(* Logix 5000 project; controller CarbonScout_MK6 vendor 1 type 14 code 154 rev 32.11; software revision 32.00; part 10 of 17 *)
(* tags used below, declared in another part *)
   Delay : TIMER;
   ExtraValveCNTReached : BOOL;
   i : DINT;
   LIT_Prev : REAL;
   LocalSampleTank : DINT;
   ONS : BOOL[32];
   TankDiagnosticCheck : BOOL;
   TimeCompare : TimerCompare;
   XRF_DirtyWinCounter : COUNTER;
   AI_FIT_01 : P_AIn;   // Purge water flow
   AI_LIT_01 : P_AIn;   // Carbon Scout Laser Level Transmitter
   AI_LIT_02 : P_AIn;   // Carbon Scout Cone Level Transmitter
   AI_PIT_01 : P_AIn;   // Water supply pressure
   CS_Alarms : P_Alarm[80];
   CS_DINTParams : DINT[100];
   CS_REALParams : REAL[80];   // CS REAL Parameters
   CS_Seq : GEK_Sequence;
   CS_Tank : CS_TankParams[20];
   CS_Timer : TIMER[80];
   CS_XRF : XRF;
   NetworkHealthy : DINT;
   Oneshot : DINT;
   Oneshot3 : DINT;
   TimeAndDate : DINT[7];
   Valve_SPR_01_Stats : GekkoValveStat;
   Valve_XV_01_Stats : GekkoValveStat;
   Valve_XV_02_Stats : GekkoValveStat;
   Valve_XV_03_Stats : GekkoValveStat;
   Valve_XV_04_Stats : GekkoValveStat;
   Valve_XV_05_Stats : GekkoValveStat;
   Valve_XV_06_Stats : GekkoValveStat;
   Valve_XV_07_Stats : GekkoValveStat;
   Valve_XV_08_Stats : GekkoValveStat;
   Valve_XV_09_Stats : GekkoValveStat;
   Valve_XV_10_Stats : GekkoValveStat;
   Valve_XV_11 : P_ValveSO;   // Purge Valve
   Valve_XV_11_Stats : GekkoValveStat;
   Valve_XV_12 : P_ValveSO;   // Slurry inlet vavle
   Valve_XV_12_Stats : GekkoValveStat;
   Valve_XV_13_Stats : GekkoValveStat;
   Valve_XV_14 : P_ValveSO;   // Top wash vavle
   Valve_XV_14_Stats : GekkoValveStat;
   Valve_XV_15_Stats : GekkoValveStat;
   Valve_XV_16_Stats : GekkoValveStat;
   Valve_XV_17 : P_ValveSO;   // Sample cone outlet vavle
   Valve_XV_17_Stats : GekkoValveStat;
   Valve_XV_18_Stats : GekkoValveStat;
   Valve_XV_19 : P_ValveSO;   // Laser window
   Valve_XV_19_Stats : GekkoValveStat;
   Valve_XV_21_30_Stats : GekkoValveStat;
   Valve_XV_30_Stats : GekkoValveStat;
   XRF_RAWDINT : DINT[100];
(* SeqProgram, continued *)

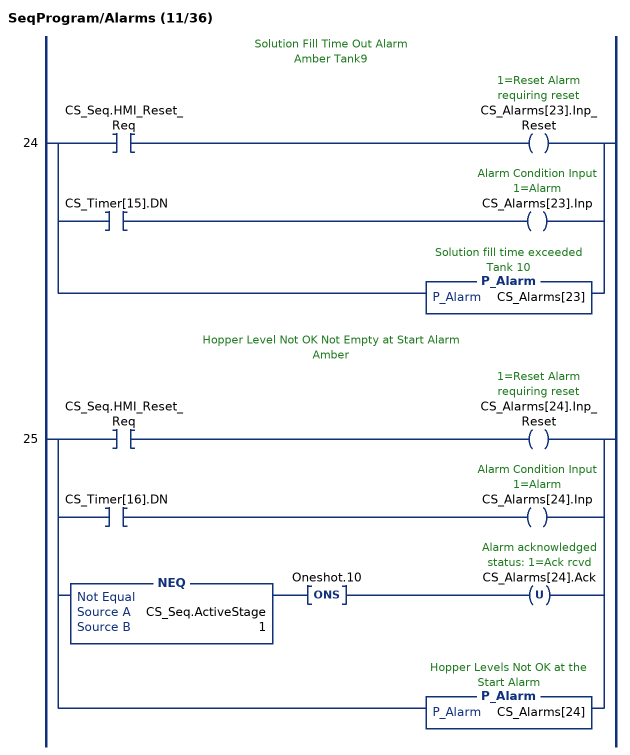
   // Solution Fill Time Out Alarm
   // Amber Tank9
   24: [XIC(CS_Seq.HMI_Reset_Req) OTE(CS_Alarms[23].Inp_Reset) ,XIC(CS_Timer[15].DN) OTE(CS_Alarms[23].Inp) ,P_Alarm(CS_Alarms[23]) ];
   // Hopper Level Not OK Not Empty at Start Alarm
   // Amber
   25: [XIC(CS_Seq.HMI_Reset_Req) OTE(CS_Alarms[24].Inp_Reset) ,XIC(CS_Timer[16].DN) OTE(CS_Alarms[24].Inp) ,NEQ(CS_Seq.ActiveStage,1) ONS(Oneshot.10) OTU(CS_Alarms[24].Ack) ,P_Alarm(CS_Alarms[24]) ];
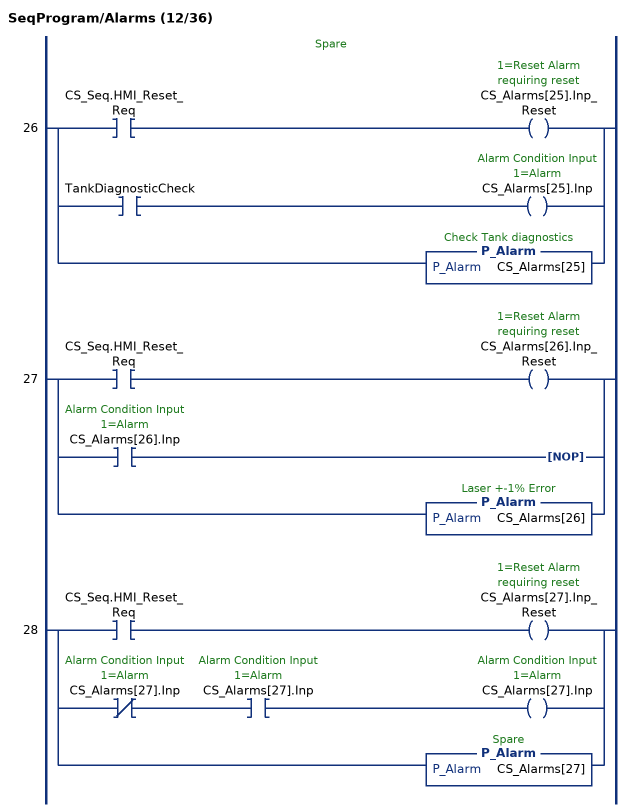
   // Spare
   26: [XIC(CS_Seq.HMI_Reset_Req) OTE(CS_Alarms[25].Inp_Reset) ,XIC(TankDiagnosticCheck) OTE(CS_Alarms[25].Inp) ,P_Alarm(CS_Alarms[25]) ];
   27: [XIC(CS_Seq.HMI_Reset_Req) OTE(CS_Alarms[26].Inp_Reset) ,XIC(CS_Alarms[26].Inp) NOP() ,P_Alarm(CS_Alarms[26]) ];
   28: [XIC(CS_Seq.HMI_Reset_Req) OTE(CS_Alarms[27].Inp_Reset) ,XIO(CS_Alarms[27].Inp) XIC(CS_Alarms[27].Inp) OTE(CS_Alarms[27].Inp) ,P_Alarm(CS_Alarms[27]) ];
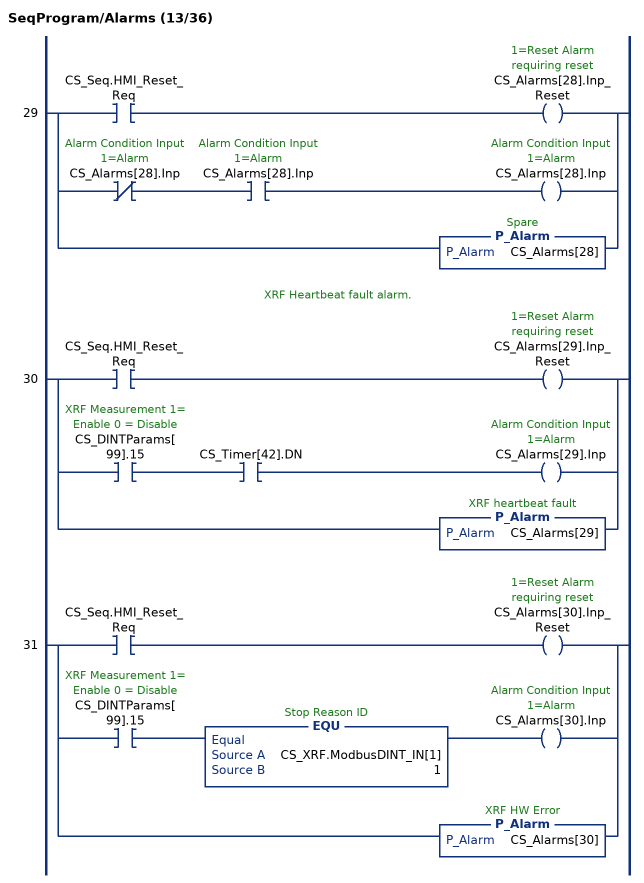
   29: [XIC(CS_Seq.HMI_Reset_Req) OTE(CS_Alarms[28].Inp_Reset) ,XIO(CS_Alarms[28].Inp) XIC(CS_Alarms[28].Inp) OTE(CS_Alarms[28].Inp) ,P_Alarm(CS_Alarms[28]) ];
   // XRF Heartbeat fault alarm.
   30: [XIC(CS_Seq.HMI_Reset_Req) OTE(CS_Alarms[29].Inp_Reset) ,XIC(CS_DINTParams[99].15) XIC(CS_Timer[42].DN) OTE(CS_Alarms[29].Inp) ,P_Alarm(CS_Alarms[29]) ];
   31: [XIC(CS_Seq.HMI_Reset_Req) OTE(CS_Alarms[30].Inp_Reset) ,XIC(CS_DINTParams[99].15) EQU(CS_XRF.ModbusDINT_IN[1],1) OTE(CS_Alarms[30].Inp) ,P_Alarm(CS_Alarms[30]) ];
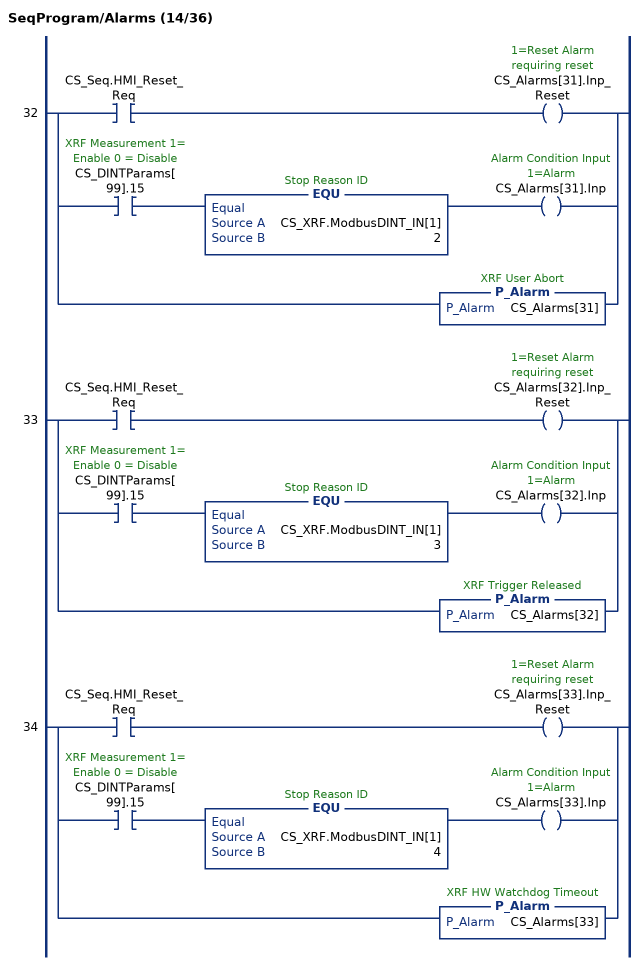
   32: [XIC(CS_Seq.HMI_Reset_Req) OTE(CS_Alarms[31].Inp_Reset) ,XIC(CS_DINTParams[99].15) EQU(CS_XRF.ModbusDINT_IN[1],2) OTE(CS_Alarms[31].Inp) ,P_Alarm(CS_Alarms[31]) ];
   33: [XIC(CS_Seq.HMI_Reset_Req) OTE(CS_Alarms[32].Inp_Reset) ,XIC(CS_DINTParams[99].15) EQU(CS_XRF.ModbusDINT_IN[1],3) OTE(CS_Alarms[32].Inp) ,P_Alarm(CS_Alarms[32]) ];
   34: [XIC(CS_Seq.HMI_Reset_Req) OTE(CS_Alarms[33].Inp_Reset) ,XIC(CS_DINTParams[99].15) EQU(CS_XRF.ModbusDINT_IN[1],4) OTE(CS_Alarms[33].Inp) ,P_Alarm(CS_Alarms[33]) ];
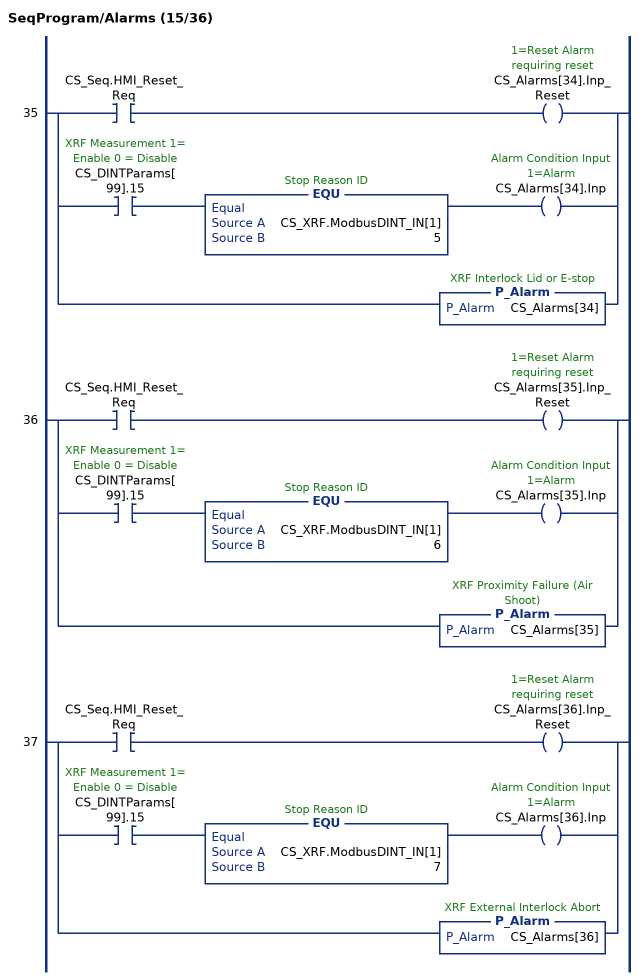
   35: [XIC(CS_Seq.HMI_Reset_Req) OTE(CS_Alarms[34].Inp_Reset) ,XIC(CS_DINTParams[99].15) EQU(CS_XRF.ModbusDINT_IN[1],5) OTE(CS_Alarms[34].Inp) ,P_Alarm(CS_Alarms[34]) ];
   36: [XIC(CS_Seq.HMI_Reset_Req) OTE(CS_Alarms[35].Inp_Reset) ,XIC(CS_DINTParams[99].15) EQU(CS_XRF.ModbusDINT_IN[1],6) OTE(CS_Alarms[35].Inp) ,P_Alarm(CS_Alarms[35]) ];
   37: [XIC(CS_Seq.HMI_Reset_Req) OTE(CS_Alarms[36].Inp_Reset) ,XIC(CS_DINTParams[99].15) EQU(CS_XRF.ModbusDINT_IN[1],7) OTE(CS_Alarms[36].Inp) ,P_Alarm(CS_Alarms[36]) ];
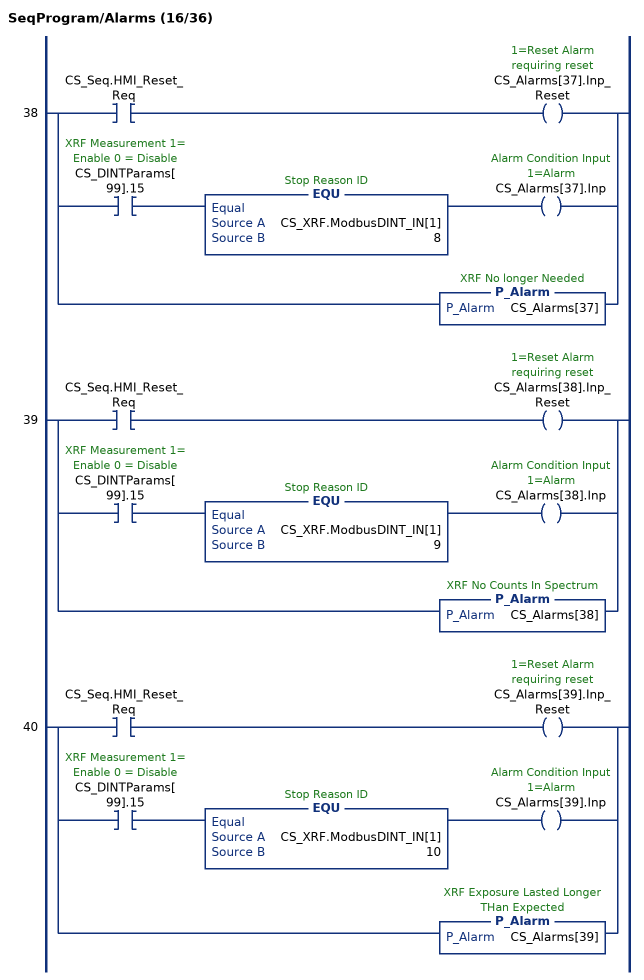
   38: [XIC(CS_Seq.HMI_Reset_Req) OTE(CS_Alarms[37].Inp_Reset) ,XIC(CS_DINTParams[99].15) EQU(CS_XRF.ModbusDINT_IN[1],8) OTE(CS_Alarms[37].Inp) ,P_Alarm(CS_Alarms[37]) ];
   39: [XIC(CS_Seq.HMI_Reset_Req) OTE(CS_Alarms[38].Inp_Reset) ,XIC(CS_DINTParams[99].15) EQU(CS_XRF.ModbusDINT_IN[1],9) OTE(CS_Alarms[38].Inp) ,P_Alarm(CS_Alarms[38]) ];
   40: [XIC(CS_Seq.HMI_Reset_Req) OTE(CS_Alarms[39].Inp_Reset) ,XIC(CS_DINTParams[99].15) EQU(CS_XRF.ModbusDINT_IN[1],10) OTE(CS_Alarms[39].Inp) ,P_Alarm(CS_Alarms[39]) ];
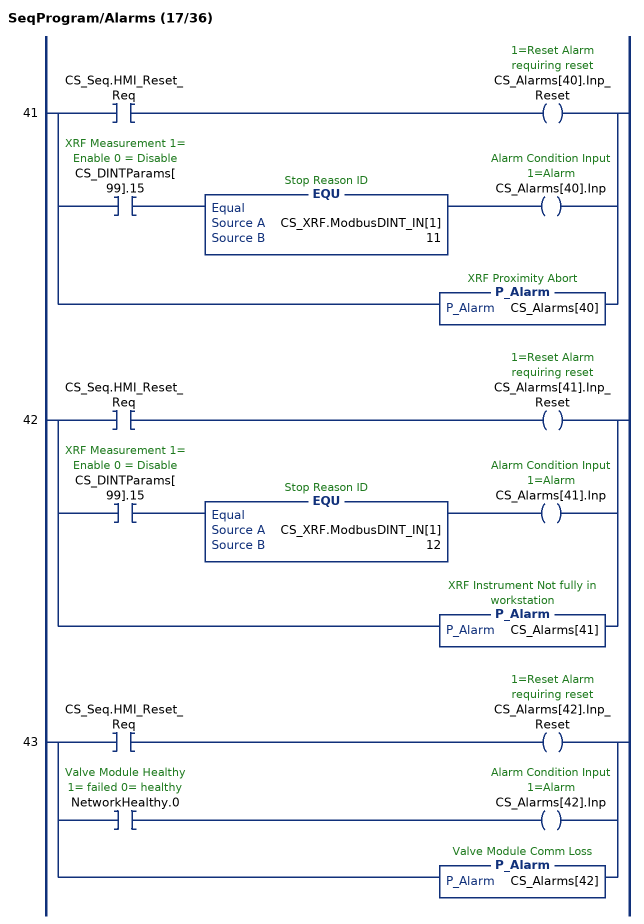
   41: [XIC(CS_Seq.HMI_Reset_Req) OTE(CS_Alarms[40].Inp_Reset) ,XIC(CS_DINTParams[99].15) EQU(CS_XRF.ModbusDINT_IN[1],11) OTE(CS_Alarms[40].Inp) ,P_Alarm(CS_Alarms[40]) ];
   42: [XIC(CS_Seq.HMI_Reset_Req) OTE(CS_Alarms[41].Inp_Reset) ,XIC(CS_DINTParams[99].15) EQU(CS_XRF.ModbusDINT_IN[1],12) OTE(CS_Alarms[41].Inp) ,P_Alarm(CS_Alarms[41]) ];
   43: [XIC(CS_Seq.HMI_Reset_Req) OTE(CS_Alarms[42].Inp_Reset) ,XIC(NetworkHealthy.0) OTE(CS_Alarms[42].Inp) ,P_Alarm(CS_Alarms[42]) ];
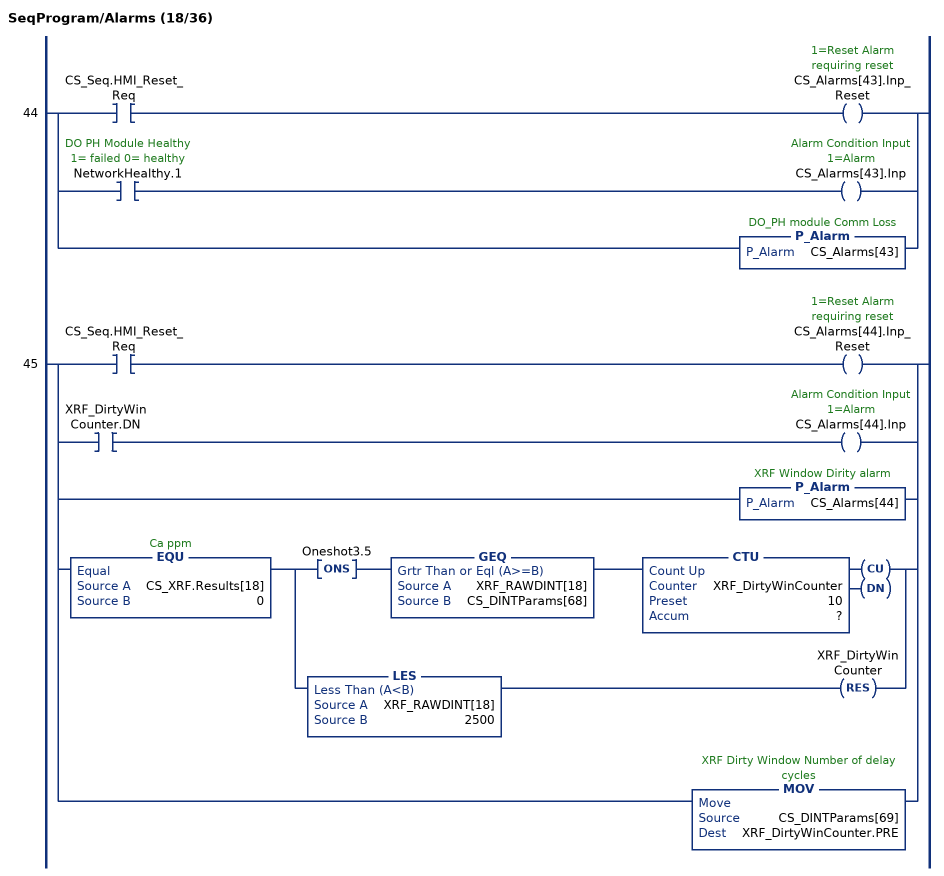
   44: [XIC(CS_Seq.HMI_Reset_Req) OTE(CS_Alarms[43].Inp_Reset) ,XIC(NetworkHealthy.1) OTE(CS_Alarms[43].Inp) ,P_Alarm(CS_Alarms[43]) ];
   45: [XIC(CS_Seq.HMI_Reset_Req) OTE(CS_Alarms[44].Inp_Reset) ,XIC(XRF_DirtyWinCounter.DN) OTE(CS_Alarms[44].Inp) ,P_Alarm(CS_Alarms[44]) ,EQU(CS_XRF.Results[18],0) [ONS(Oneshot3.5) GEQ(XRF_RAWDINT[18],CS_DINTParams[68]) CTU(XRF_DirtyWinCounter,?,?) ,LES(XRF_RAWDINT[18],2500) RES(XRF_DirtyWinCounter) ] ,MOV(CS_DINTParams[69],XRF_DirtyWinCounter.PRE) ];
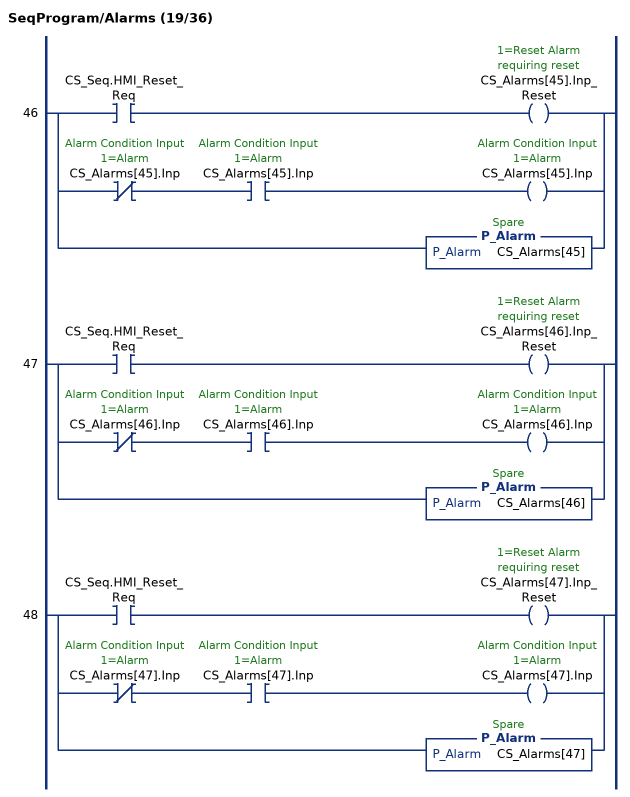
   46: [XIC(CS_Seq.HMI_Reset_Req) OTE(CS_Alarms[45].Inp_Reset) ,XIO(CS_Alarms[45].Inp) XIC(CS_Alarms[45].Inp) OTE(CS_Alarms[45].Inp) ,P_Alarm(CS_Alarms[45]) ];
   47: [XIC(CS_Seq.HMI_Reset_Req) OTE(CS_Alarms[46].Inp_Reset) ,XIO(CS_Alarms[46].Inp) XIC(CS_Alarms[46].Inp) OTE(CS_Alarms[46].Inp) ,P_Alarm(CS_Alarms[46]) ];
   48: [XIC(CS_Seq.HMI_Reset_Req) OTE(CS_Alarms[47].Inp_Reset) ,XIO(CS_Alarms[47].Inp) XIC(CS_Alarms[47].Inp) OTE(CS_Alarms[47].Inp) ,P_Alarm(CS_Alarms[47]) ];
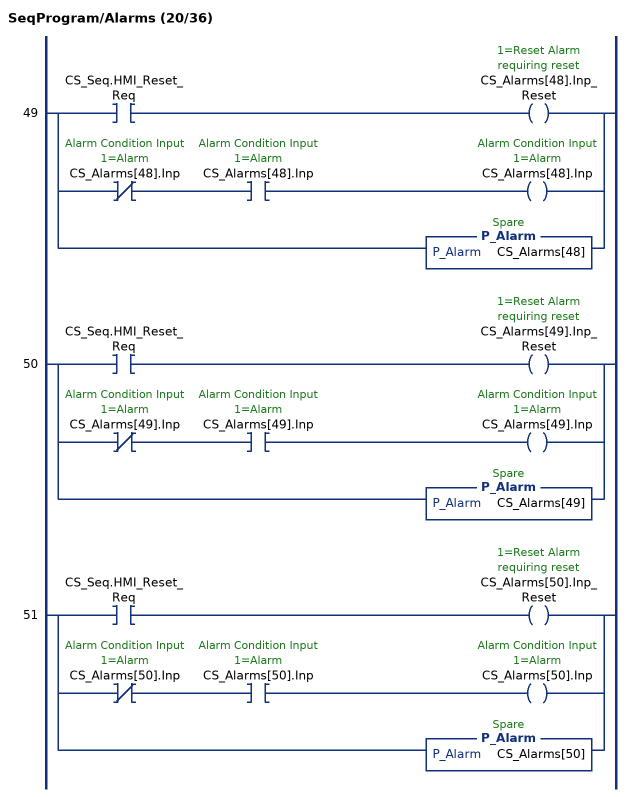
   49: [XIC(CS_Seq.HMI_Reset_Req) OTE(CS_Alarms[48].Inp_Reset) ,XIO(CS_Alarms[48].Inp) XIC(CS_Alarms[48].Inp) OTE(CS_Alarms[48].Inp) ,P_Alarm(CS_Alarms[48]) ];
   50: [XIC(CS_Seq.HMI_Reset_Req) OTE(CS_Alarms[49].Inp_Reset) ,XIO(CS_Alarms[49].Inp) XIC(CS_Alarms[49].Inp) OTE(CS_Alarms[49].Inp) ,P_Alarm(CS_Alarms[49]) ];
   51: [XIC(CS_Seq.HMI_Reset_Req) OTE(CS_Alarms[50].Inp_Reset) ,XIO(CS_Alarms[50].Inp) XIC(CS_Alarms[50].Inp) OTE(CS_Alarms[50].Inp) ,P_Alarm(CS_Alarms[50]) ];
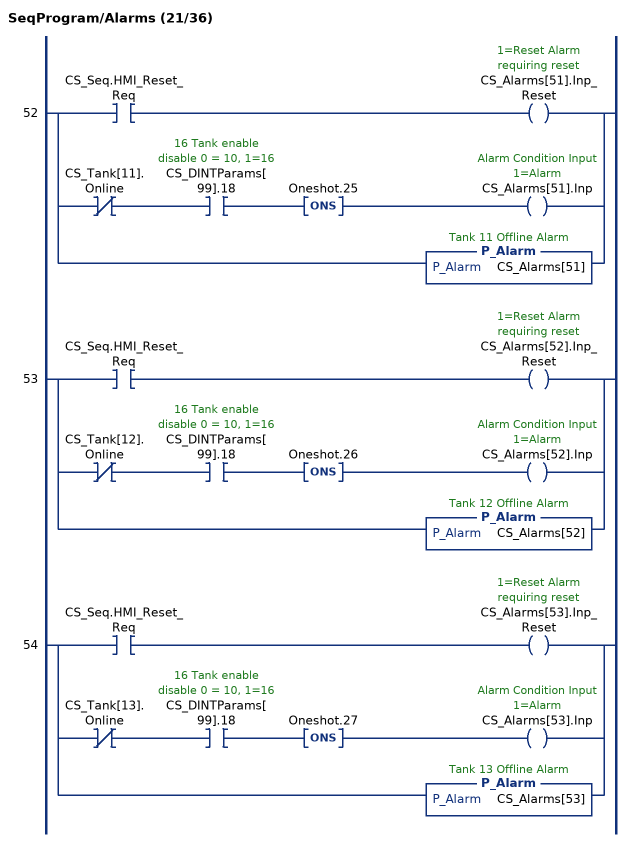
   52: [XIC(CS_Seq.HMI_Reset_Req) OTE(CS_Alarms[51].Inp_Reset) ,XIO(CS_Tank[11].Online) XIC(CS_DINTParams[99].18) ONS(Oneshot.25) OTE(CS_Alarms[51].Inp) ,P_Alarm(CS_Alarms[51]) ];
   53: [XIC(CS_Seq.HMI_Reset_Req) OTE(CS_Alarms[52].Inp_Reset) ,XIO(CS_Tank[12].Online) XIC(CS_DINTParams[99].18) ONS(Oneshot.26) OTE(CS_Alarms[52].Inp) ,P_Alarm(CS_Alarms[52]) ];
   54: [XIC(CS_Seq.HMI_Reset_Req) OTE(CS_Alarms[53].Inp_Reset) ,XIO(CS_Tank[13].Online) XIC(CS_DINTParams[99].18) ONS(Oneshot.27) OTE(CS_Alarms[53].Inp) ,P_Alarm(CS_Alarms[53]) ];
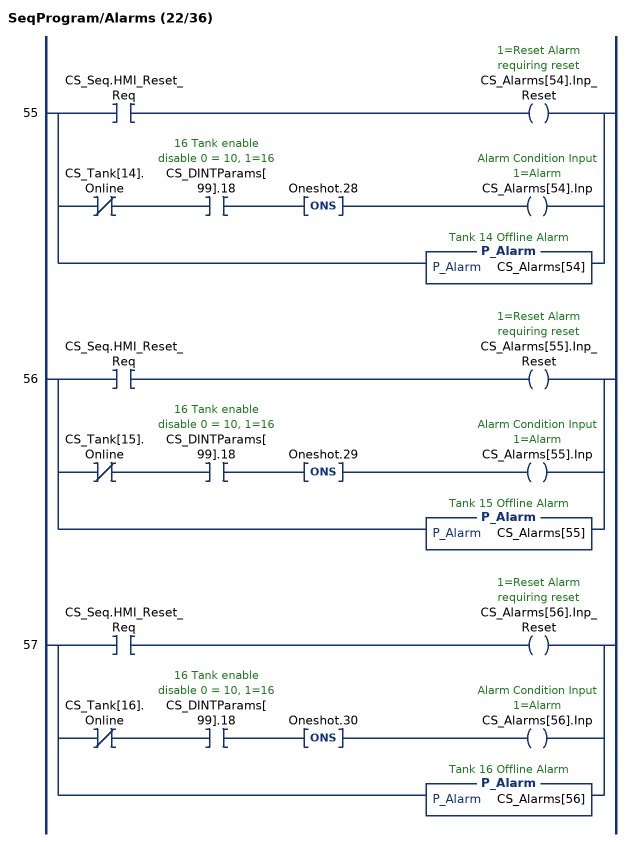
   55: [XIC(CS_Seq.HMI_Reset_Req) OTE(CS_Alarms[54].Inp_Reset) ,XIO(CS_Tank[14].Online) XIC(CS_DINTParams[99].18) ONS(Oneshot.28) OTE(CS_Alarms[54].Inp) ,P_Alarm(CS_Alarms[54]) ];
   56: [XIC(CS_Seq.HMI_Reset_Req) OTE(CS_Alarms[55].Inp_Reset) ,XIO(CS_Tank[15].Online) XIC(CS_DINTParams[99].18) ONS(Oneshot.29) OTE(CS_Alarms[55].Inp) ,P_Alarm(CS_Alarms[55]) ];
   57: [XIC(CS_Seq.HMI_Reset_Req) OTE(CS_Alarms[56].Inp_Reset) ,XIO(CS_Tank[16].Online) XIC(CS_DINTParams[99].18) ONS(Oneshot.30) OTE(CS_Alarms[56].Inp) ,P_Alarm(CS_Alarms[56]) ];
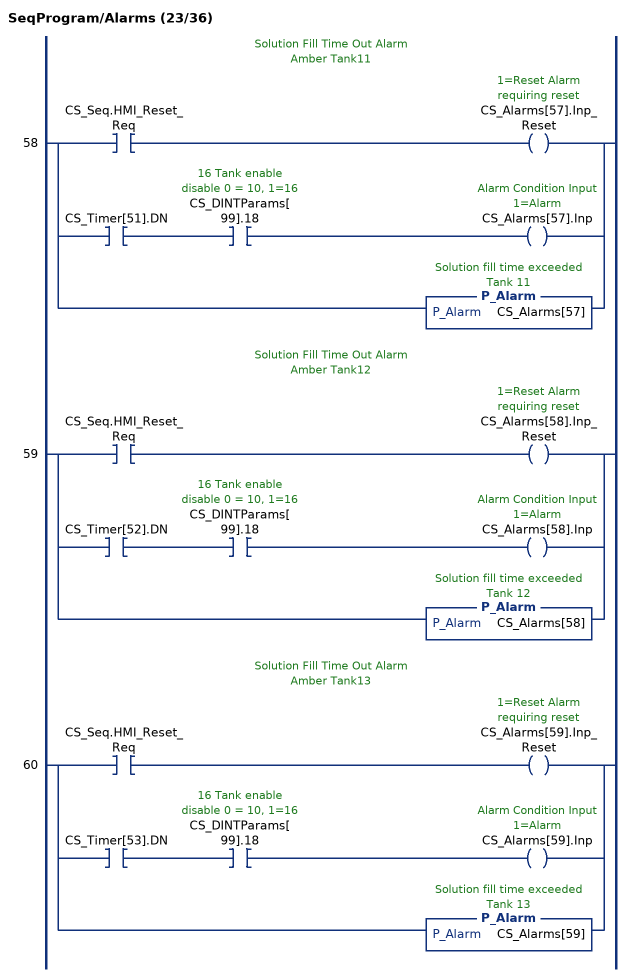
   // Solution Fill Time Out Alarm
   // Amber Tank11
   58: [XIC(CS_Seq.HMI_Reset_Req) OTE(CS_Alarms[57].Inp_Reset) ,XIC(CS_Timer[51].DN) XIC(CS_DINTParams[99].18) OTE(CS_Alarms[57].Inp) ,P_Alarm(CS_Alarms[57]) ];
   // Solution Fill Time Out Alarm
   // Amber Tank12
   59: [XIC(CS_Seq.HMI_Reset_Req) OTE(CS_Alarms[58].Inp_Reset) ,XIC(CS_Timer[52].DN) XIC(CS_DINTParams[99].18) OTE(CS_Alarms[58].Inp) ,P_Alarm(CS_Alarms[58]) ];
   // Solution Fill Time Out Alarm
   // Amber Tank13
   60: [XIC(CS_Seq.HMI_Reset_Req) OTE(CS_Alarms[59].Inp_Reset) ,XIC(CS_Timer[53].DN) XIC(CS_DINTParams[99].18) OTE(CS_Alarms[59].Inp) ,P_Alarm(CS_Alarms[59]) ];
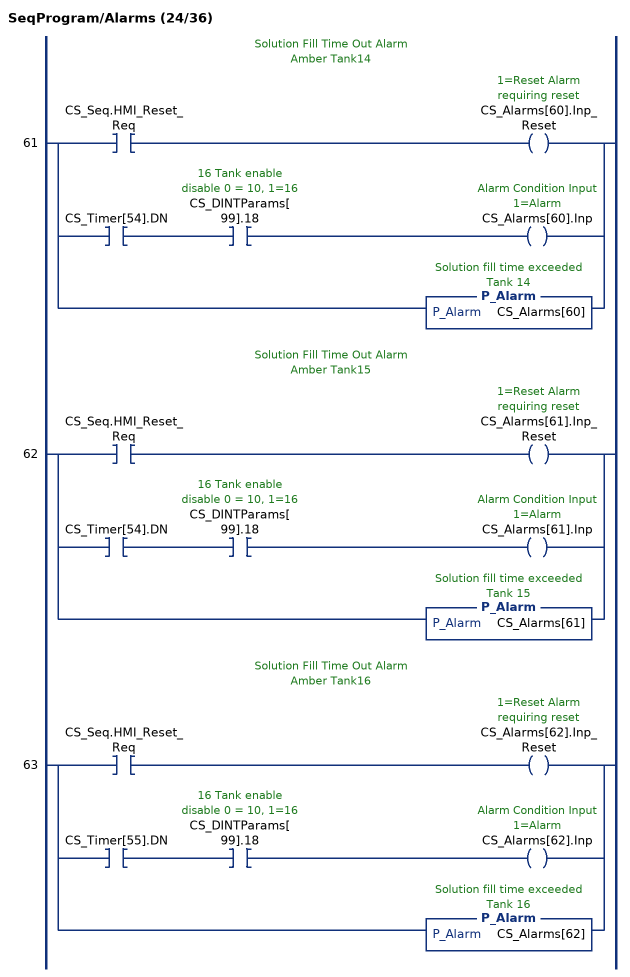
   // Solution Fill Time Out Alarm
   // Amber Tank14
   61: [XIC(CS_Seq.HMI_Reset_Req) OTE(CS_Alarms[60].Inp_Reset) ,XIC(CS_Timer[54].DN) XIC(CS_DINTParams[99].18) OTE(CS_Alarms[60].Inp) ,P_Alarm(CS_Alarms[60]) ];
   // Solution Fill Time Out Alarm
   // Amber Tank15
   62: [XIC(CS_Seq.HMI_Reset_Req) OTE(CS_Alarms[61].Inp_Reset) ,XIC(CS_Timer[54].DN) XIC(CS_DINTParams[99].18) OTE(CS_Alarms[61].Inp) ,P_Alarm(CS_Alarms[61]) ];
   // Solution Fill Time Out Alarm
   // Amber Tank16
   63: [XIC(CS_Seq.HMI_Reset_Req) OTE(CS_Alarms[62].Inp_Reset) ,XIC(CS_Timer[55].DN) XIC(CS_DINTParams[99].18) OTE(CS_Alarms[62].Inp) ,P_Alarm(CS_Alarms[62]) ];
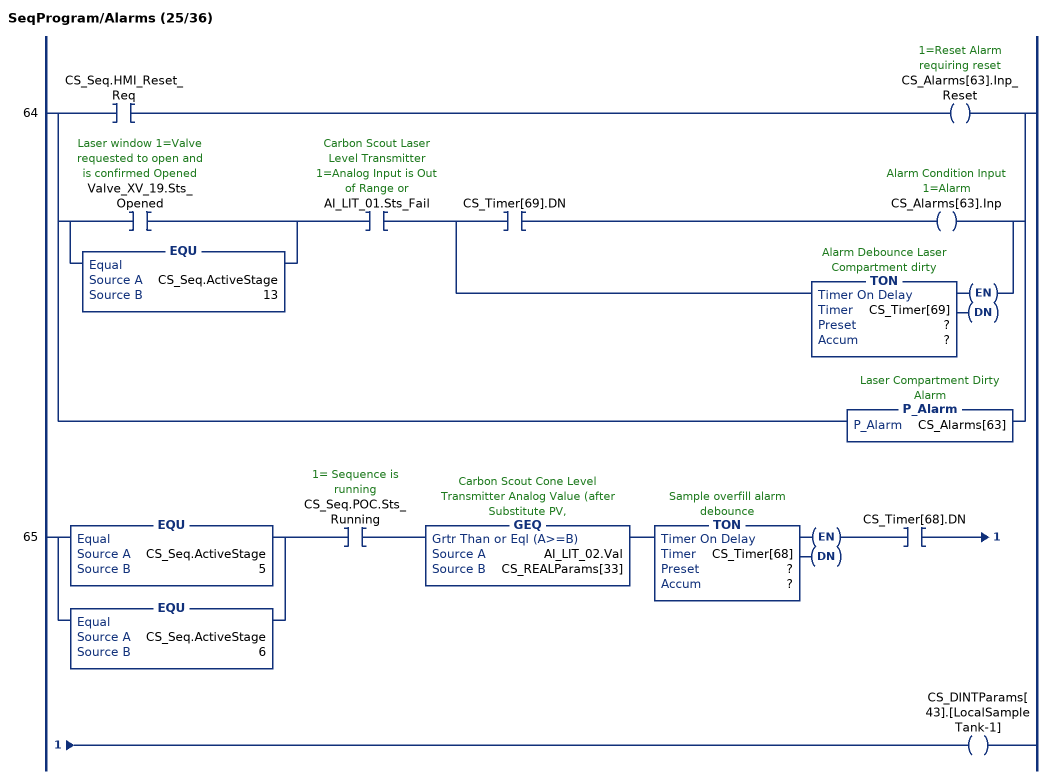
   64: [XIC(CS_Seq.HMI_Reset_Req) OTE(CS_Alarms[63].Inp_Reset) ,[XIC(Valve_XV_19.Sts_Opened) ,EQU(CS_Seq.ActiveStage,13) ] XIC(AI_LIT_01.Sts_Fail) [XIC(CS_Timer[69].DN) OTE(CS_Alarms[63].Inp) ,TON(CS_Timer[69],?,?) ] ,P_Alarm(CS_Alarms[63]) ];
   65: [EQU(CS_Seq.ActiveStage,5) ,EQU(CS_Seq.ActiveStage,6) ]XIC(CS_Seq.POC.Sts_Running)GEQ(AI_LIT_02.Val,CS_REALParams[33])TON(CS_Timer[68],?,?)XIC(CS_Timer[68].DN)OTE(CS_DINTParams[43].[LocalSampleTank-1]);
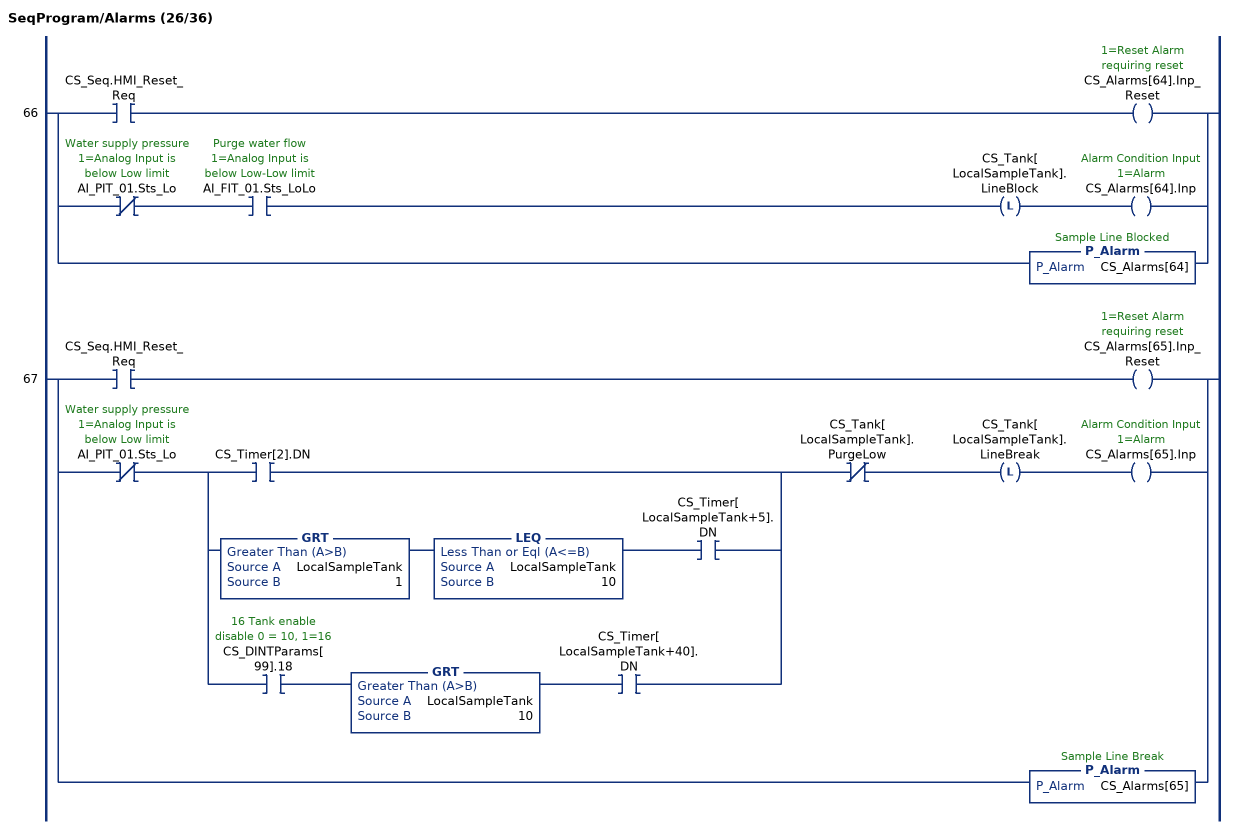
   66: [XIC(CS_Seq.HMI_Reset_Req) OTE(CS_Alarms[64].Inp_Reset) ,XIO(AI_PIT_01.Sts_Lo) XIC(AI_FIT_01.Sts_LoLo) OTL(CS_Tank[LocalSampleTank].LineBlock) OTE(CS_Alarms[64].Inp) ,P_Alarm(CS_Alarms[64]) ];
   67: [XIC(CS_Seq.HMI_Reset_Req) OTE(CS_Alarms[65].Inp_Reset) ,XIO(AI_PIT_01.Sts_Lo) [XIC(CS_Timer[2].DN) ,GRT(LocalSampleTank,1) LEQ(LocalSampleTank,10) XIC(CS_Timer[LocalSampleTank+5].DN) ,XIC(CS_DINTParams[99].18) GRT(LocalSampleTank,10) XIC(CS_Timer[LocalSampleTank+40].DN) ] XIO(CS_Tank[LocalSampleTank].PurgeLow) OTL(CS_Tank[LocalSampleTank].LineBreak) OTE(CS_Alarms[65].Inp) ,P_Alarm(CS_Alarms[65]) ];
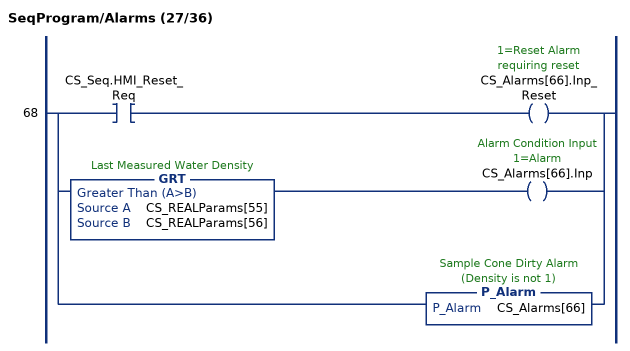
   68: [XIC(CS_Seq.HMI_Reset_Req) OTE(CS_Alarms[66].Inp_Reset) ,GRT(CS_REALParams[55],CS_REALParams[56]) OTE(CS_Alarms[66].Inp) ,P_Alarm(CS_Alarms[66]) ];
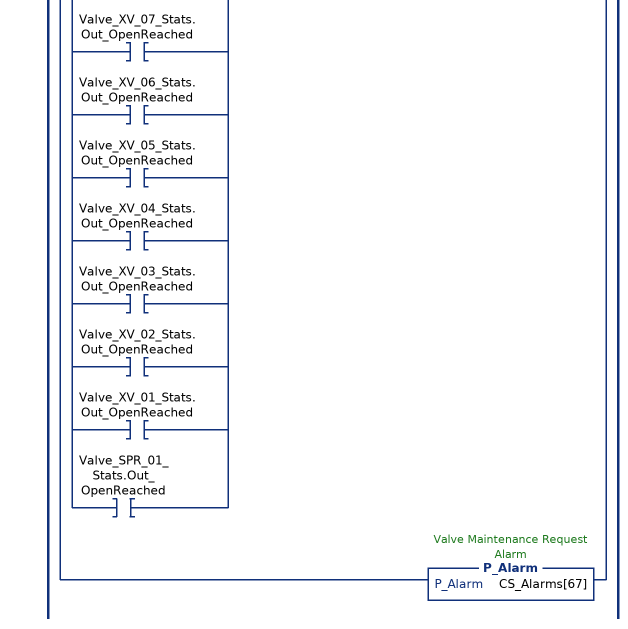
   69: [XIC(CS_Seq.HMI_Reset_Req) OTE(CS_Alarms[67].Inp_Reset) ,[XIC(Valve_XV_30_Stats.Out_OpenReached) ,XIC(ExtraValveCNTReached) ,XIC(Valve_XV_21_30_Stats.Out_OpenReached) ,XIC(Valve_XV_19_Stats.Out_OpenReached) ,XIC(Valve_XV_18_Stats.Out_OpenReached) ,XIC(Valve_XV_17_Stats.Out_OpenReached) ,XIC(Valve_XV_16_Stats.Out_OpenReached) ,XIC(Valve_XV_15_Stats.Out_OpenReached) ,XIC(Valve_XV_14_Stats.Out_OpenReached) ,XIC(Valve_XV_13_Stats.Out_OpenReached) ,XIC(Valve_XV_12_Stats.Out_OpenReached) ,XIC(Valve_XV_11_Stats.Out_OpenReached) ,XIC(Valve_XV_10_Stats.Out_OpenReached) ,XIC(Valve_XV_09_Stats.Out_OpenReached) ,XIC(Valve_XV_08_Stats.Out_OpenReached) ,XIC(Valve_XV_07_Stats.Out_OpenReached) ,XIC(Valve_XV_06_Stats.Out_OpenReached) ,XIC(Valve_XV_05_Stats.Out_OpenReached) ,XIC(Valve_XV_04_Stats.Out_OpenReached) ,XIC(Valve_XV_03_Stats.Out_OpenReached) ,XIC(Valve_XV_02_Stats.Out_OpenReached) ,XIC(Valve_XV_01_Stats.Out_OpenReached) ,XIC(Valve_SPR_01_Stats.Out_OpenReached) ] OTE(CS_Alarms[67].Inp) ,P_Alarm(CS_Alarms[67]) ];
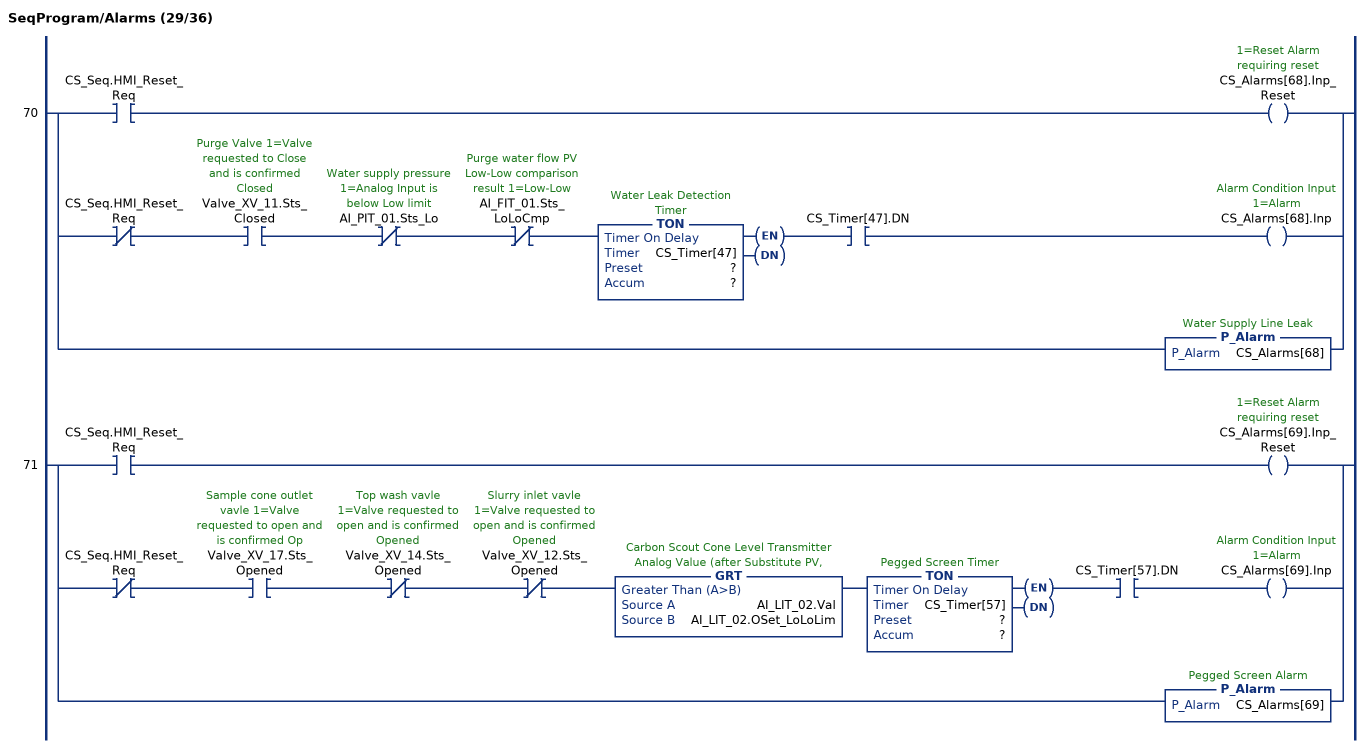
   70: [XIC(CS_Seq.HMI_Reset_Req) OTE(CS_Alarms[68].Inp_Reset) ,XIO(CS_Seq.HMI_Reset_Req) XIC(Valve_XV_11.Sts_Closed) XIO(AI_PIT_01.Sts_Lo) XIO(AI_FIT_01.Sts_LoLoCmp) TON(CS_Timer[47],?,?) XIC(CS_Timer[47].DN) OTE(CS_Alarms[68].Inp) ,P_Alarm(CS_Alarms[68]) ];
   71: [XIC(CS_Seq.HMI_Reset_Req) OTE(CS_Alarms[69].Inp_Reset) ,XIO(CS_Seq.HMI_Reset_Req) XIC(Valve_XV_17.Sts_Opened) XIO(Valve_XV_14.Sts_Opened) XIO(Valve_XV_12.Sts_Opened) GRT(AI_LIT_02.Val,AI_LIT_02.OSet_LoLoLim) TON(CS_Timer[57],?,?) XIC(CS_Timer[57].DN) OTE(CS_Alarms[69].Inp) ,P_Alarm(CS_Alarms[69]) ];
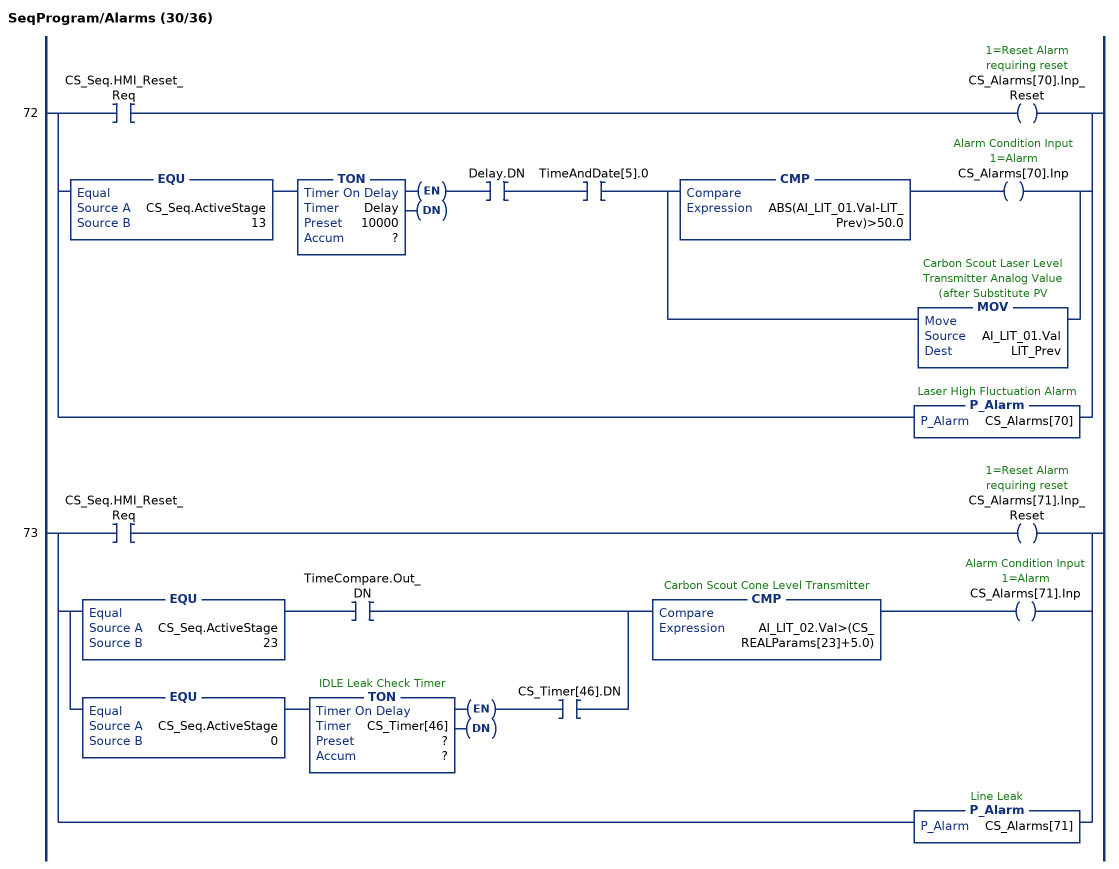
   72: [XIC(CS_Seq.HMI_Reset_Req) OTE(CS_Alarms[70].Inp_Reset) ,EQU(CS_Seq.ActiveStage,13) TON(Delay,?,?) XIC(Delay.DN) XIC(TimeAndDate[5].0) [CMP(ABS(AI_LIT_01.Val-LIT_Prev)>50.0) OTE(CS_Alarms[70].Inp) ,MOV(AI_LIT_01.Val,LIT_Prev) ] ,P_Alarm(CS_Alarms[70]) ];
   73: [XIC(CS_Seq.HMI_Reset_Req) OTE(CS_Alarms[71].Inp_Reset) ,[EQU(CS_Seq.ActiveStage,23) XIC(TimeCompare.Out_DN) ,EQU(CS_Seq.ActiveStage,0) TON(CS_Timer[46],?,?) XIC(CS_Timer[46].DN) ] CMP(AI_LIT_02.Val>(CS_REALParams[23]+5.0)) OTE(CS_Alarms[71].Inp) ,P_Alarm(CS_Alarms[71]) ];
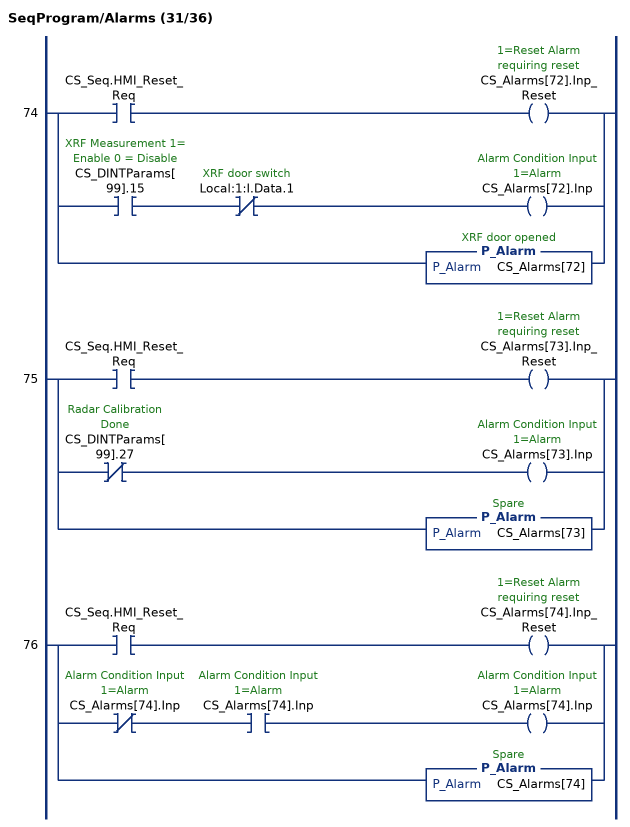
   74: [XIC(CS_Seq.HMI_Reset_Req) OTE(CS_Alarms[72].Inp_Reset) ,XIC(CS_DINTParams[99].15) XIO(Local:1:I.Data.1) OTE(CS_Alarms[72].Inp) ,P_Alarm(CS_Alarms[72]) ];
   75: [XIC(CS_Seq.HMI_Reset_Req) OTE(CS_Alarms[73].Inp_Reset) ,XIO(CS_DINTParams[99].27) OTE(CS_Alarms[73].Inp) ,P_Alarm(CS_Alarms[73]) ];
   76: [XIC(CS_Seq.HMI_Reset_Req) OTE(CS_Alarms[74].Inp_Reset) ,XIO(CS_Alarms[74].Inp) XIC(CS_Alarms[74].Inp) OTE(CS_Alarms[74].Inp) ,P_Alarm(CS_Alarms[74]) ];
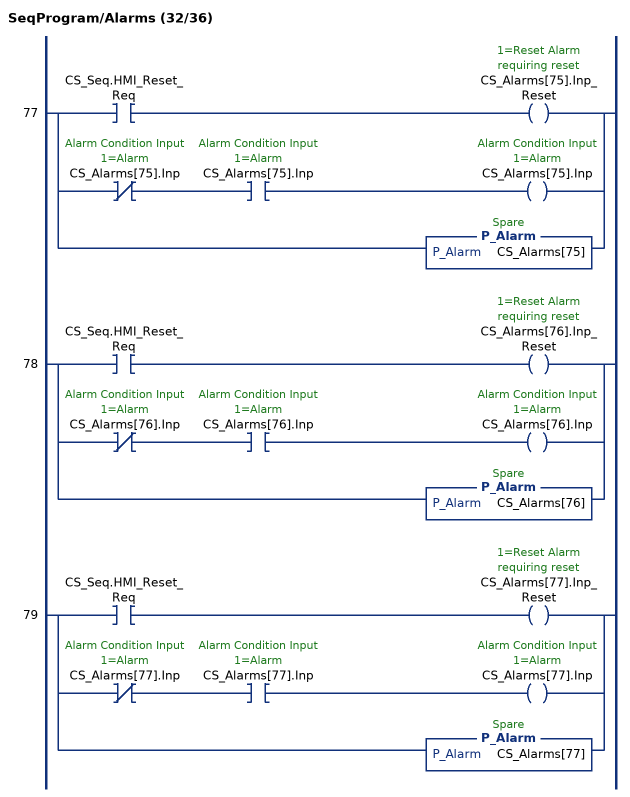
   77: [XIC(CS_Seq.HMI_Reset_Req) OTE(CS_Alarms[75].Inp_Reset) ,XIO(CS_Alarms[75].Inp) XIC(CS_Alarms[75].Inp) OTE(CS_Alarms[75].Inp) ,P_Alarm(CS_Alarms[75]) ];
   78: [XIC(CS_Seq.HMI_Reset_Req) OTE(CS_Alarms[76].Inp_Reset) ,XIO(CS_Alarms[76].Inp) XIC(CS_Alarms[76].Inp) OTE(CS_Alarms[76].Inp) ,P_Alarm(CS_Alarms[76]) ];
   79: [XIC(CS_Seq.HMI_Reset_Req) OTE(CS_Alarms[77].Inp_Reset) ,XIO(CS_Alarms[77].Inp) XIC(CS_Alarms[77].Inp) OTE(CS_Alarms[77].Inp) ,P_Alarm(CS_Alarms[77]) ];
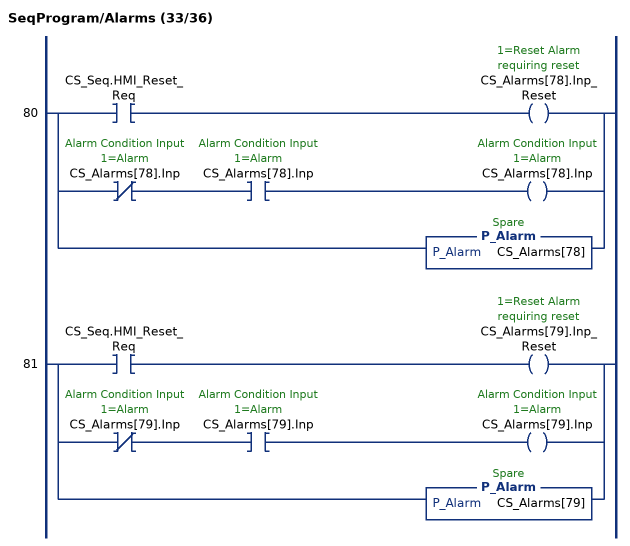
   80: [XIC(CS_Seq.HMI_Reset_Req) OTE(CS_Alarms[78].Inp_Reset) ,XIO(CS_Alarms[78].Inp) XIC(CS_Alarms[78].Inp) OTE(CS_Alarms[78].Inp) ,P_Alarm(CS_Alarms[78]) ];
   81: [XIC(CS_Seq.HMI_Reset_Req) OTE(CS_Alarms[79].Inp_Reset) ,XIO(CS_Alarms[79].Inp) XIC(CS_Alarms[79].Inp) OTE(CS_Alarms[79].Inp) ,P_Alarm(CS_Alarms[79]) ];
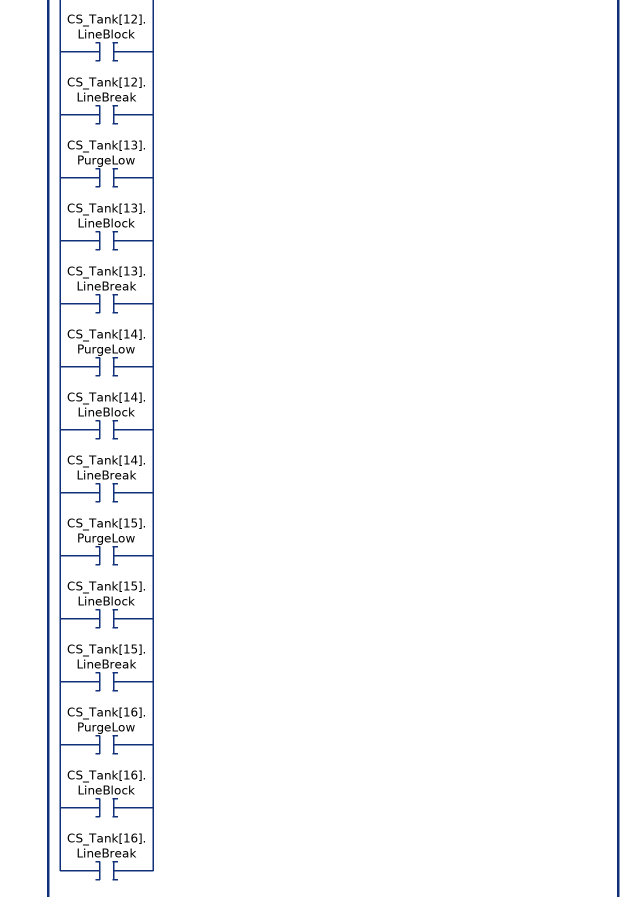
   82: [XIC(CS_Tank[1].PurgeLow) ,XIC(CS_Tank[1].LineBlock) ,XIC(CS_Tank[1].LineBreak) ,XIC(CS_Tank[2].PurgeLow) ,XIC(CS_Tank[2].LineBlock) ,XIC(CS_Tank[2].LineBreak) ,XIC(CS_Tank[3].PurgeLow) ,XIC(CS_Tank[3].LineBlock) ,XIC(CS_Tank[3].LineBreak) ,XIC(CS_Tank[4].PurgeLow) ,XIC(CS_Tank[4].LineBlock) ,XIC(CS_Tank[4].LineBreak) ,XIC(CS_Tank[5].PurgeLow) ,XIC(CS_Tank[5].LineBlock) ,XIC(CS_Tank[5].LineBreak) ,XIC(CS_Tank[6].PurgeLow) ,XIC(CS_Tank[6].LineBlock) ,XIC(CS_Tank[6].LineBreak) ,XIC(CS_Tank[7].PurgeLow) ,XIC(CS_Tank[7].LineBlock) ,XIC(CS_Tank[7].LineBreak) ,XIC(CS_Tank[8].PurgeLow) ,XIC(CS_Tank[8].LineBlock) ,XIC(CS_Tank[8].LineBreak) ,XIC(CS_Tank[9].PurgeLow) ,XIC(CS_Tank[9].LineBlock) ,XIC(CS_Tank[9].LineBreak) ,XIC(CS_Tank[10].PurgeLow) ,XIC(CS_Tank[10].LineBlock) ,XIC(CS_Tank[10].LineBreak) ,XIC(CS_Tank[11].PurgeLow) ,XIC(CS_Tank[11].LineBlock) ,XIC(CS_Tank[11].LineBreak) ,XIC(CS_Tank[12].PurgeLow) ,XIC(CS_Tank[12].LineBlock) ,XIC(CS_Tank[12].LineBreak) ,XIC(CS_Tank[13].PurgeLow) ,XIC(CS_Tank[13].LineBlock) ,XIC(CS_Tank[13].LineBreak) ,XIC(CS_Tank[14].PurgeLow) ,XIC(CS_Tank[14].LineBlock) ,XIC(CS_Tank[14].LineBreak) ,XIC(CS_Tank[15].PurgeLow) ,XIC(CS_Tank[15].LineBlock) ,XIC(CS_Tank[15].LineBreak) ,XIC(CS_Tank[16].PurgeLow) ,XIC(CS_Tank[16].LineBlock) ,XIC(CS_Tank[16].LineBreak) ]OTE(TankDiagnosticCheck);
